{attribute 'qualified_only'}
VAR_GLOBAL
END_VAR

(* stored: Version 1.1.0.1, ProductVersion 3.1.4024.10
   GVL GVL_Recipe: Id {d24cf871-76b1-4e56-93c1-b4eae84cd2b4} *)
